(* PLC project Unnamed, Actility iec61131 1.x.x *)
(* stored: creationDateTime 2013-03-22T14:32:43, version 1.x.x, modificationDateTime 2013-03-22T14:32:43 *)

CONFIGURATION config
  RESOURCE resource1 ON PLC
  END_RESOURCE
END_CONFIGURATION
